FUNCTION_BLOCK FB_CalcFocalLengthLensSet EXTENDS FB_Fallible IMPLEMENTS I_CalcFocalLengthLensSet
VAR
    iConvertUnits : I_ConvertUnitsLREAL;
    iLensCompounder : I_LensCompounder;
    iCalcFocalLengthSingleLens : I_CalcFocalLengthSingleLens;

    fbLens : FB_Lens;
    fbFocalLengthLens : FB_QuantityLREALPublic(Units := 'm');

    {attribute 'pytmc' := 'pv: FocalLength'}
    fbFocalLength : FB_QuantityLREALPublic(Units := 'm');

    nIndex : INT;
END_VAR


METHOD Calculate
VAR_INPUT
    LensSet : I_LensSet;
END_VAR
VAR_IN_OUT
    FocalLength : FB_QuantityLREALPublic(Units := 'm');
END_VAR

ClearError();

SetUnits(Units := FocalLength.Units);

// Check for an invalid lens set input.
IF LensSet.GetError() THEN
    SetError(
        Msg := CONCAT('The input lens set has the following error message: [',
        CONCAT(LensSet.GetErrorMsg(),
        ']'))
    );
    FocalLength.SetError(Msg := GetErrorMsg());
    RETURN;
END_IF

// Check for an invalid number of lenses
IF LensSet.NumLenses < 1.0 THEN
    SetError(
        Msg := CONCAT('The input lens set has 0 or negative lenses: [',
        CONCAT(INT_TO_STRING(LensSet.NumLenses),
        ']'))
    );
    FocalLength.SetError(Msg := GetErrorMsg());
    RETURN;
END_IF

// Check for a number of lenses greater than the max.
IF LensSet.NumLenses > GVL_Physics.nMaxNumLensesInSet THEN
    SetError(
        Msg := CONCAT('The input lens set number of lenses is greater than the global max number: [',
        CONCAT(INT_TO_STRING(LensSet.NumLenses),
        CONCAT('] = (setting) > (max) = [',
        CONCAT(INT_TO_STRING(GVL_Physics.nMaxNumLensesInSet),
        ']'))))
    );
    FocalLength.SetError(Msg := GetErrorMsg());
    RETURN;
END_IF

iLensCompounder.Reset();

FOR nIndex := 1 TO LensSet.NumLenses BY 1 DO
    LensSet.GetLens(
        LensNum := nIndex,
        Lens := fbLens
    );

    IF LensSet.GetError() THEN
        SetError(
            Msg := CONCAT('The lens set returned the following error message when attempting to get a lens: [',
            CONCAT(LensSet.GetErrorMsg(),
            ']'))
        );
        FocalLength.SetError(Msg := GetErrorMsg());
        RETURN;
    END_IF

    iCalcFocalLengthSingleLens.Calculate(
        Lens := fbLens,
        FocalLength := fbFocalLengthLens
    );

    IF iCalcFocalLengthSingleLens.GetError() THEN
        SetError(Msg :=
            CONCAT('Error returned when attempting the calculate focal length for lens number: [',
            CONCAT(INT_TO_STRING(nIndex),
            CONCAT(']. Error message is: ',
            iCalcFocalLengthSingleLens.GetErrorMsg())))
        );
        RETURN;
    END_IF

    iLensCompounder.Compound(
        FocalLength := fbFocalLengthLens,
        Multiplier := fbLens.Multiplier,
        FocalLengthCompounded := fbFocalLength
    );

    // Check for an error while compounding lenses.
    IF iLensCompounder.GetError() THEN
        SetError(
            Msg := CONCAT('Error detected while compounding lenses: [',
            CONCAT(iLensCompounder.GetErrorMsg(),
            ']'))
        );
        FocalLength.SetError(Msg := GetErrorMsg());
        RETURN;
    END_IF
END_FOR

FocalLength := fbFocalLength;
END_METHOD


METHOD PROTECTED ClearError

SUPER^.ClearError();

fbFocalLength.ClearError();
END_METHOD


METHOD FB_init : BOOL
VAR_INPUT
    bInitRetains : BOOL; // if TRUE, the retain variables are initialized (warm start / cold start)
    bInCopyCode : BOOL;  // if TRUE, the instance afterwards gets moved into the copy code (online change)

    ConvertUnits : I_ConvertUnitsLREAL;
    LensCompounder : I_LensCompounder;
    CalcFocalLengthSingleLens : I_CalcFocalLengthSingleLens;
END_VAR

THIS^.iConvertUnits := ConvertUnits;
THIS^.iLensCompounder := LensCompounder;
THIS^.iCalcFocalLengthSingleLens := CalcFocalLengthSingleLens;
END_METHOD


METHOD PROTECTED SetError
VAR_INPUT
    Msg : T_MaxString;
END_VAR

SUPER^.SetError(Msg := Msg);

fbFocalLength.SetError(Msg := Msg);
END_METHOD


METHOD PRIVATE SetUnits
VAR_INPUT
    Units : T_MaxString;
END_VAR

fbFocalLengthLens.Units := Units;
fbFocalLength.Units := Units;
END_METHOD

END_FUNCTION_BLOCK

(* stored: Version 1.1.0.1
   POU FB_CalcFocalLengthLensSet: Id {6543ad7e-352c-476d-a708-9a7e07f74363}, SpecialFunc None
   Method Calculate: Id {f5016e8c-13ab-47cb-a173-def6706fd2c4}
   Method ClearError: Id {85feb07e-790f-4b47-bebd-7692a9984a0d}
   Method FB_init: Id {1f20d000-d2a9-49d0-af13-4ff4a0f34aef}
   Method SetError: Id {5f27a043-9969-438c-a750-7a002bbe0e22}
   Method SetUnits: Id {7e175d42-711c-49a0-a07a-db592521747b} *)
